# EPICS SNL sequencer program: dxp/branches/R3-0-branch/dxpApp/src/dxpMED.st
program dxpMED("P=13GE2:med:,DXP=dxp,MCA=mca,N_DETECTORS=16")

/*  This sequencer program works with dxp.db and dxpMED.db.
 *  It supports Copying PVs from the first DXP to all of the DXPs
 *  and multi-element MCA operations
 *
 *  Mark Rivers
 *  January 7, 2005
 *
 * This program must be compiled with the recursive option so that multiple copies
 * can run at once */
option +r;

/* Allow the program to start, even if not all assigned channels are connected.
 * This could be useful if dxpMED is running on a different ioc. */
option -c;

%%#include <stdlib.h>
%%#include <errlog.h>

#define MAX_DETECTORS 100
#define MAX_SCAS 16
/* MAX_ROIS must be defined as MAX_DETECTORS * MAX_SCAS.
   It can't be done in SNL because of syntax limitations. */
#define MAX_ROIS 1600

int i;
int j;
int k;
int chan;
int det;
int nDetectors;
int prevAcquiring;
int allDone;
char temp[100];

char *prefix;
char *dxp;
char *mca;

double  TriggerPeakingTime[MAX_DETECTORS];
assign  TriggerPeakingTime to {"","","","","","","","","","","","","","","","",
                       "","","","","","","","","","","","","","","",""};
int     CopyTriggerPeakingTime; assign CopyTriggerPeakingTime to "{P}CopyTriggerPeakingTime";
monitor CopyTriggerPeakingTime; evflag CopyTriggerPeakingTimeMon; sync CopyTriggerPeakingTime CopyTriggerPeakingTimeMon;

double  TriggerGapTime[MAX_DETECTORS];
assign  TriggerGapTime to {"","","","","","","","","","","","","","","","",
                        "","","","","","","","","","","","","","","",""};
int     CopyTriggerGapTime; assign CopyTriggerGapTime to "{P}CopyTriggerGapTime";
monitor CopyTriggerGapTime; evflag CopyTriggerGapTimeMon; sync CopyTriggerGapTime CopyTriggerGapTimeMon;

double  TriggerThreshold[MAX_DETECTORS];
assign  TriggerThreshold to {"","","","","","","","","","","","","","","","",
                      "","","","","","","","","","","","","","","",""};
int     CopyTriggerThreshold; assign CopyTriggerThreshold to "{P}CopyTriggerThreshold";
monitor CopyTriggerThreshold; evflag CopyTriggerThresholdMon; sync CopyTriggerThreshold CopyTriggerThresholdMon;

double  PeakingTime[MAX_DETECTORS];
assign  PeakingTime to {"","","","","","","","","","","","","","","","",
                  "","","","","","","","","","","","","","","",""};
int     CopyPeakingTime; assign CopyPeakingTime to "{P}CopyPeakingTime";
monitor CopyPeakingTime; evflag CopyPeakingTimeMon; sync CopyPeakingTime CopyPeakingTimeMon;

double  GapTime[MAX_DETECTORS];
assign  GapTime to {"","","","","","","","","","","","","","","","",
                   "","","","","","","","","","","","","","","",""};
int     CopyGapTime; assign CopyGapTime to "{P}CopyGapTime";
monitor CopyGapTime; evflag CopyGapTimeMon; sync CopyGapTime CopyGapTimeMon;

double  EnergyThreshold[MAX_DETECTORS];
assign  EnergyThreshold to {"","","","","","","","","","","","","","","","",
                      "","","","","","","","","","","","","","","",""};
int     CopyEnergyThreshold; assign CopyEnergyThreshold to "{P}CopyEnergyThreshold";
monitor CopyEnergyThreshold; evflag CopyEnergyThresholdMon; sync CopyEnergyThreshold CopyEnergyThresholdMon;

double  MaxWidth[MAX_DETECTORS];
assign  MaxWidth to {"","","","","","","","","","","","","","","","",
                      "","","","","","","","","","","","","","","",""};
int     CopyMaxWidth; assign CopyMaxWidth to "{P}CopyMaxWidth";
monitor CopyMaxWidth; evflag CopyMaxWidthMon; sync CopyMaxWidth CopyMaxWidthMon;

double  BaselineCutPercent[MAX_DETECTORS];
assign  BaselineCutPercent to {"","","","","","","","","","","","","","","","",
                         "","","","","","","","","","","","","","","",""};
int     CopyBaselineCutPercent; assign CopyBaselineCutPercent to "{P}CopyBaselineCutPercent";
monitor CopyBaselineCutPercent; evflag CopyBaselineCutPercentMon; sync CopyBaselineCutPercent CopyBaselineCutPercentMon;

double  BaselineCutEnable[MAX_DETECTORS];
assign  BaselineCutEnable to {"","","","","","","","","","","","","","","","",
                          "","","","","","","","","","","","","","","",""};
int     CopyBaselineCutEnable; assign CopyBaselineCutEnable to "{P}CopyBaselineCutEnable";
monitor CopyBaselineCutEnable; evflag CopyBaselineCutEnableMon; sync CopyBaselineCutEnable CopyBaselineCutEnableMon;

double  BaselineThreshold[MAX_DETECTORS];
assign  BaselineThreshold to {"","","","","","","","","","","","","","","","",
                        "","","","","","","","","","","","","","","",""};
int     CopyBaselineThreshold; assign CopyBaselineThreshold to "{P}CopyBaselineThreshold";
monitor CopyBaselineThreshold; evflag CopyBaselineThresholdMon; sync CopyBaselineThreshold CopyBaselineThresholdMon;

double  BaselineFilterLength[MAX_DETECTORS];
assign  BaselineFilterLength to {"","","","","","","","","","","","","","","","",
                     "","","","","","","","","","","","","","","",""};
int     CopyBaselineFilterLength; assign CopyBaselineFilterLength to "{P}CopyBaselineFilterLength";
monitor CopyBaselineFilterLength; evflag CopyBaselineFilterLengthMon; sync CopyBaselineFilterLength CopyBaselineFilterLengthMon;

double  PreampGain[MAX_DETECTORS];
assign  PreampGain to {"","","","","","","","","","","","","","","","",
                  "","","","","","","","","","","","","","","",""};
int     CopyPreampGain; assign CopyPreampGain to "{P}CopyPreampGain";
monitor CopyPreampGain; evflag CopyPreampGainMon; sync CopyPreampGain CopyPreampGainMon;

double  MaxEnergy[MAX_DETECTORS];
assign  MaxEnergy to {"","","","","","","","","","","","","","","","",
                 "","","","","","","","","","","","","","","",""};
int     CopyMaxEnergy; assign CopyMaxEnergy to "{P}CopyMaxEnergy";
monitor CopyMaxEnergy; evflag CopyMaxEnergyMon; sync CopyMaxEnergy CopyMaxEnergyMon;

double  ADCPercentRule[MAX_DETECTORS];
assign  ADCPercentRule to {"","","","","","","","","","","","","","","","",
                     "","","","","","","","","","","","","","","",""};
int     CopyADCPercentRule; assign CopyADCPercentRule to "{P}CopyADCPercentRule";
monitor CopyADCPercentRule; evflag CopyADCPercentRuleMon; sync CopyADCPercentRule CopyADCPercentRuleMon;

/*int     ReadDXP[MAX_DETECTORS];  */
/*assign  ReadDXP to {"","","","","","","","","","","","","","","","", */
/*                    "","","","","","","","","","","","","","","",""}; */
/*int     ReadDXPs; assign ReadDXPs to "{P}DoReadDXPs"; */
/*monitor ReadDXPs; evflag ReadDXPsMon; sync ReadDXPs ReadDXPsMon; */

int     ReadBaselineHistogram[MAX_DETECTORS];
assign  ReadBaselineHistogram to {"","","","","","","","","","","","","","","","",
                            "","","","","","","","","","","","","","","",""};
int     ReadBaselineHistograms; assign ReadBaselineHistograms to "{P}DoReadBaselineHistograms";
monitor ReadBaselineHistograms; evflag ReadBaselineHistogramsMon; sync ReadBaselineHistograms ReadBaselineHistogramsMon;

int     ReadTrace[MAX_DETECTORS];
assign  ReadTrace to {"","","","","","","","","","","","","","","","",
                         "","","","","","","","","","","","","","","",""};
int     ReadTraces; assign ReadTraces to "{P}DoReadTraces";
monitor ReadTraces; evflag ReadTracesMon; sync ReadTraces ReadTracesMon;

double  TraceTime[MAX_DETECTORS];
assign  TraceTime to {"","","","","","","","","","","","","","","","",
                         "","","","","","","","","","","","","","","",""};
double  TraceTimes; assign TraceTimes to "{P}TraceTimes";
monitor TraceTimes; evflag TraceTimesMon; sync TraceTimes TraceTimesMon;

int     TraceMode[MAX_DETECTORS];
assign  TraceMode to {"","","","","","","","","","","","","","","","",
                         "","","","","","","","","","","","","","","",""};
int     TraceModes; assign TraceModes to "{P}TraceModes";
monitor TraceModes; evflag TraceModesMon; sync TraceModes TraceModesMon;

int     ReadMCA[MAX_DETECTORS];
assign  ReadMCA to {"","","","","","","","","","","","","","","","",
                    "","","","","","","","","","","","","","","",""};
int     ReadMCAs; assign ReadMCAs to "{P}DoReadAll";
monitor ReadMCAs; evflag ReadMCAsMon; sync ReadMCAs ReadMCAsMon;
int     ReadMCAAll; assign ReadMCAAll to "";

int     statusMCA[MAX_DETECTORS];
assign  statusMCA to {"","","","","","","","","","","","","","","","",
                      "","","","","","","","","","","","","","","",""};
int     StatusMCAs; assign StatusMCAs to "{P}DoStatusAll";
monitor StatusMCAs; evflag StatusMCAsMon; sync StatusMCAs StatusMCAsMon;
int     statusMCAAll; assign statusMCAAll to "";

int     mcaAcquiring[MAX_DETECTORS];
assign  mcaAcquiring to {"","","","","","","","","","","","","","","","",
                         "","","","","","","","","","","","","","","",""};
monitor mcaAcquiring; evflag  mcaAcquiringMon; sync mcaAcquiring mcaAcquiringMon;
int     Acquiring; assign Acquiring to "";
monitor Acquiring; evflag AcquiringMon; sync Acquiring AcquiringMon;

double  mcaPresetReal[MAX_DETECTORS];
assign  mcaPresetReal to {"","","","","","","","","","","","","","","","",
                          "","","","","","","","","","","","","","","",""};
double  PresetReal; assign PresetReal to "{P}PresetReal";
monitor PresetReal; evflag PresetRealMon; sync PresetReal PresetRealMon;

double  mcaPresetLive[MAX_DETECTORS];
assign  mcaPresetLive to {"","","","","","","","","","","","","","","","",
                          "","","","","","","","","","","","","","","",""};
double  PresetLive; assign PresetLive to "{P}PresetLive";
monitor PresetLive; evflag PresetLiveMon; sync PresetLive PresetLiveMon;

double  mcaDeadTime[MAX_DETECTORS];
assign  mcaDeadTime to {"","","","","","","","","","","","","","","","",
                        "","","","","","","","","","","","","","","",""};
double  DeadTime; assign DeadTime to "{P}DeadTime";
evflag  DeadTimeMon; sync mcaDeadTime DeadTimeMon;

int     mcaROILow[MAX_ROIS];
assign  mcaROILow to {"","","","","","","","","","","","","","","","",
                      "","","","","","","","","","","","","","","","",
                      "","","","","","","","","","","","","","","","",
                      "","","","","","","","","","","","","","","","",
                      "","","","","","","","","","","","","","","","",
                      "","","","","","","","","","","","","","","","",
                      "","","","","","","","","","","","","","","","",
                      "","","","","","","","","","","","","","","","",
                      "","","","","","","","","","","","","","","","",
                      "","","","","","","","","","","","","","","","",
                      "","","","","","","","","","","","","","","","",
                      "","","","","","","","","","","","","","","","",
                      "","","","","","","","","","","","","","","","",
                      "","","","","","","","","","","","","","","","",
                      "","","","","","","","","","","","","","","","",
                      "","","","","","","","","","","","","","","","",
                      "","","","","","","","","","","","","","","","",
                      "","","","","","","","","","","","","","","","",
                      "","","","","","","","","","","","","","","","",
                      "","","","","","","","","","","","","","","","",
                      "","","","","","","","","","","","","","","","",
                      "","","","","","","","","","","","","","","","",
                      "","","","","","","","","","","","","","","","",
                      "","","","","","","","","","","","","","","","",
                      "","","","","","","","","","","","","","","","",
                      "","","","","","","","","","","","","","","","",
                      "","","","","","","","","","","","","","","","",
                      "","","","","","","","","","","","","","","","",
                      "","","","","","","","","","","","","","","","",
                      "","","","","","","","","","","","","","","","",
                      "","","","","","","","","","","","","","","","",
                      "","","","","","","","","","","","","","","",""};
monitor mcaROILow; evflag  mcaROILowMon; sync mcaROILow mcaROILowMon;

int    mcaROIHigh[MAX_ROIS];
assign mcaROIHigh to {"","","","","","","","","","","","","","","","",
                      "","","","","","","","","","","","","","","","",
                      "","","","","","","","","","","","","","","","",
                      "","","","","","","","","","","","","","","","",
                      "","","","","","","","","","","","","","","","",
                      "","","","","","","","","","","","","","","","",
                      "","","","","","","","","","","","","","","","",
                      "","","","","","","","","","","","","","","","",
                      "","","","","","","","","","","","","","","","",
                      "","","","","","","","","","","","","","","","",
                      "","","","","","","","","","","","","","","","",
                      "","","","","","","","","","","","","","","","",
                      "","","","","","","","","","","","","","","","",
                      "","","","","","","","","","","","","","","","",
                      "","","","","","","","","","","","","","","","",
                      "","","","","","","","","","","","","","","","",
                      "","","","","","","","","","","","","","","","",
                      "","","","","","","","","","","","","","","","",
                      "","","","","","","","","","","","","","","","",
                      "","","","","","","","","","","","","","","","",
                      "","","","","","","","","","","","","","","","",
                      "","","","","","","","","","","","","","","","",
                      "","","","","","","","","","","","","","","","",
                      "","","","","","","","","","","","","","","","",
                      "","","","","","","","","","","","","","","","",
                      "","","","","","","","","","","","","","","","",
                      "","","","","","","","","","","","","","","","",
                      "","","","","","","","","","","","","","","","",
                      "","","","","","","","","","","","","","","","",
                      "","","","","","","","","","","","","","","","",
                      "","","","","","","","","","","","","","","","",
                      "","","","","","","","","","","","","","","",""};
monitor mcaROIHigh; evflag  mcaROIHighMon; sync mcaROIHigh mcaROIHighMon;

int     dxpSCALow[MAX_ROIS];
assign  dxpSCALow to {"","","","","","","","","","","","","","","","",
                      "","","","","","","","","","","","","","","","",
                      "","","","","","","","","","","","","","","","",
                      "","","","","","","","","","","","","","","","",
                      "","","","","","","","","","","","","","","","",
                      "","","","","","","","","","","","","","","","",
                      "","","","","","","","","","","","","","","","",
                      "","","","","","","","","","","","","","","","",
                      "","","","","","","","","","","","","","","","",
                      "","","","","","","","","","","","","","","","",
                      "","","","","","","","","","","","","","","","",
                      "","","","","","","","","","","","","","","","",
                      "","","","","","","","","","","","","","","","",
                      "","","","","","","","","","","","","","","","",
                      "","","","","","","","","","","","","","","","",
                      "","","","","","","","","","","","","","","","",
                      "","","","","","","","","","","","","","","","",
                      "","","","","","","","","","","","","","","","",
                      "","","","","","","","","","","","","","","","",
                      "","","","","","","","","","","","","","","","",
                      "","","","","","","","","","","","","","","","",
                      "","","","","","","","","","","","","","","","",
                      "","","","","","","","","","","","","","","","",
                      "","","","","","","","","","","","","","","","",
                      "","","","","","","","","","","","","","","","",
                      "","","","","","","","","","","","","","","","",
                      "","","","","","","","","","","","","","","","",
                      "","","","","","","","","","","","","","","","",
                      "","","","","","","","","","","","","","","","",
                      "","","","","","","","","","","","","","","","",
                      "","","","","","","","","","","","","","","","",
                      "","","","","","","","","","","","","","","",""};

int    dxpSCAHigh[MAX_ROIS];
assign dxpSCAHigh to {"","","","","","","","","","","","","","","","",
                      "","","","","","","","","","","","","","","","",
                      "","","","","","","","","","","","","","","","",
                      "","","","","","","","","","","","","","","","",
                      "","","","","","","","","","","","","","","","",
                      "","","","","","","","","","","","","","","","",
                      "","","","","","","","","","","","","","","","",
                      "","","","","","","","","","","","","","","","",
                      "","","","","","","","","","","","","","","","",
                      "","","","","","","","","","","","","","","","",
                      "","","","","","","","","","","","","","","","",
                      "","","","","","","","","","","","","","","","",
                      "","","","","","","","","","","","","","","","",
                      "","","","","","","","","","","","","","","","",
                      "","","","","","","","","","","","","","","","",
                      "","","","","","","","","","","","","","","","",
                      "","","","","","","","","","","","","","","","",
                      "","","","","","","","","","","","","","","","",
                      "","","","","","","","","","","","","","","","",
                      "","","","","","","","","","","","","","","","",
                      "","","","","","","","","","","","","","","","",
                      "","","","","","","","","","","","","","","","",
                      "","","","","","","","","","","","","","","","",
                      "","","","","","","","","","","","","","","","",
                      "","","","","","","","","","","","","","","","",
                      "","","","","","","","","","","","","","","","",
                      "","","","","","","","","","","","","","","","",
                      "","","","","","","","","","","","","","","","",
                      "","","","","","","","","","","","","","","","",
                      "","","","","","","","","","","","","","","","",
                      "","","","","","","","","","","","","","","","",
                      "","","","","","","","","","","","","","","",""};

int AcquireBusy; assign AcquireBusy to "{P}AcquireBusy";

ss dxp_control {
    state init {
        when() {
            /* We set the following event flags to force these modes and
               labels to be set correctly initially */
            prefix = macValueGet("P");
            dxp = macValueGet("DXP");
            mca = macValueGet("MCA");
            nDetectors = atoi(macValueGet("N_DETECTORS"));
            if ((nDetectors <= 0) || (nDetectors > MAX_DETECTORS)) {
              printf ("N_DETECTORS is illegal.\n");
              nDetectors = 0;
            }
            if (MAX_ROIS != (MAX_DETECTORS * MAX_SCAS)) {
              printf ("N_DETECTORS, MAX_SCAS and MAX_ROIS are inconsistent.\n");
              nDetectors = 0;
            }
            for (i=0; i<nDetectors; i++) {
               det = i+1;
               sprintf(temp, "%s%s%d:TriggerPeakingTime", prefix, dxp, det);
               pvAssign(TriggerPeakingTime[i], temp);
               sprintf(temp, "%s%s%d:TriggerGapTime", prefix, dxp, det);
               pvAssign(TriggerGapTime[i], temp);
               sprintf(temp, "%s%s%d:TriggerThreshold", prefix, dxp, det);
               pvAssign(TriggerThreshold[i], temp);
               sprintf(temp, "%s%s%d:PeakingTime", prefix, dxp, det);
               pvAssign(PeakingTime[i], temp);
               sprintf(temp, "%s%s%d:GapTime", prefix, dxp, det);
               pvAssign(GapTime[i], temp);
               sprintf(temp, "%s%s%d:EnergyThreshold", prefix, dxp, det);
               pvAssign(EnergyThreshold[i], temp);
               sprintf(temp, "%s%s%d:MaxWidth", prefix, dxp, det);
               pvAssign(MaxWidth[i], temp);
               sprintf(temp, "%s%s%d:BaselineCutPercent", prefix, dxp, det);
               pvAssign(BaselineCutPercent[i], temp);
               sprintf(temp, "%s%s%d:BaselineCutEnable", prefix, dxp, det);
               pvAssign(BaselineCutEnable[i], temp);
               sprintf(temp, "%s%s%d:BaselineThreshold", prefix, dxp, det);
               pvAssign(BaselineThreshold[i], temp);
               sprintf(temp, "%s%s%d:BaselineFilterLength", prefix, dxp, det);
               pvAssign(BaselineFilterLength[i], temp);
               sprintf(temp, "%s%s%d:PreampGain", prefix, dxp, det);
               pvAssign(PreampGain[i], temp);
               sprintf(temp, "%s%s%d:MaxEnergy", prefix, dxp, det);
               pvAssign(MaxEnergy[i], temp);
               sprintf(temp, "%s%s%d:ADCPercentRule", prefix, dxp, det);
               pvAssign(ADCPercentRule[i], temp);
/*               sprintf(temp, "%s%s%d:ReadParams.PROC", prefix, dxp, det); */
/*               pvAssign(ReadDXP[i], temp); */
               sprintf(temp, "%s%s%d:BaselineHistogram.PROC", prefix, dxp, det);
               pvAssign(ReadBaselineHistogram[i], temp);
               sprintf(temp, "%s%s%d:TraceData.PROC", prefix, dxp, det);
               pvAssign(ReadTrace[i], temp);
               sprintf(temp, "%s%s%d:TraceTime", prefix, dxp, det);
               pvAssign(TraceTime[i], temp);
               sprintf(temp, "%s%s%d:TraceMode", prefix, dxp, det);
               pvAssign(TraceMode[i], temp);
               sprintf(temp, "%s%s%d.READ", prefix, mca, det);
               pvAssign(ReadMCA[i], temp);
               sprintf(temp, "%s%s%d.PROC", prefix, mca, det);
               pvAssign(statusMCA[i], temp);
               sprintf(temp, "%s%s%d.ACQG", prefix, mca, det);
               pvAssign(mcaAcquiring[i], temp);
               sprintf(temp, "%s%s%d.PRTM", prefix, mca, det);
               pvAssign(mcaPresetReal[i], temp);
               sprintf(temp, "%s%s%d.PLTM", prefix, mca, det);
               pvAssign(mcaPresetLive[i], temp);
               sprintf(temp, "%s%s%d.IDTIM", prefix, mca, det);
               pvAssign(mcaDeadTime[i], temp);
               pvMonitor(mcaDeadTime[i]);
/*
               for (j=0; j<MAX_SCAS; j++) {
                   k = i*MAX_SCAS + j;
                   sprintf(temp, "%s%s%d.R%iLO", prefix, mca, det, j);
                   pvAssign(mcaROILow[k], temp);
                   pvMonitor(mcaROILow[k]);
                   sprintf(temp, "%s%s%d.R%iHI", prefix, mca, det, j);
                   pvAssign(mcaROIHigh[k], temp);
                   pvMonitor(mcaROIHigh[k]);
                   sprintf(temp, "%s%s%d.SCA%i_LO", prefix, dxp, det, j);
                   pvAssign(dxpSCALow[k], temp);
                   sprintf(temp, "%s%s%d.SCA%i_HI", prefix, dxp, det, j);
                   pvAssign(dxpSCAHigh[k], temp);
               }
*/
           }
           sprintf(temp, "%s%sAll.PROC", prefix, mca);
           pvAssign(statusMCAAll, temp);
           sprintf(temp, "%s%sAll.READ", prefix, mca);
           pvAssign(ReadMCAAll, temp);
           sprintf(temp, "%s%sAll.ACQG", prefix, mca);
           pvAssign(Acquiring, temp);
           prevAcquiring = Acquiring;
        } state waitConnected
    }
    state waitConnected {

        when (nDetectors <= 0) {
          printf (">>>>>>>>>>>>>> dxpMED is dead. <<<<<<<<<<<<<<\n");
        } state dead

        when (pvAssignCount () == pvConnectCount ()) {
          printf ("dxpMED: All channels connected.\n");
        } state monitor_changes

    }
    state dead {
      when (delay (3600.0)) {
      } state dead
    }

    state monitor_changes {

        when (pvAssignCount () != pvConnectCount ()) {
          printf ("dxpMED: Not all channels connected.\n");
        } state waitConnected

        when(efTestAndClear(CopyTriggerPeakingTimeMon) && (CopyTriggerPeakingTime == 1)) {
            pvGet(TriggerPeakingTime[0]);
            for (i=0; i<nDetectors; i++) {
                TriggerPeakingTime[i] = TriggerPeakingTime[0];
                pvPut(TriggerPeakingTime[i]);
            }
            CopyTriggerPeakingTime = 0;
            pvPut(CopyTriggerPeakingTime);
        } state monitor_changes

        when(efTestAndClear(CopyTriggerGapTimeMon) && (CopyTriggerGapTime == 1)) {
            pvGet(TriggerGapTime[0]);
            for (i=0; i<nDetectors; i++) {
                TriggerGapTime[i] = TriggerGapTime[0];
                pvPut(TriggerGapTime[i]);
            }
            CopyTriggerGapTime = 0;
            pvPut(CopyTriggerGapTime);
        } state monitor_changes

        when(efTestAndClear(CopyTriggerThresholdMon) && (CopyTriggerThreshold == 1)) {
            pvGet(TriggerThreshold[0]);
            for (i=0; i<nDetectors; i++) {
                TriggerThreshold[i] = TriggerThreshold[0];
                pvPut(TriggerThreshold[i]);
            }
            CopyTriggerThreshold = 0;
            pvPut(CopyTriggerThreshold);
        } state monitor_changes

        when(efTestAndClear(CopyPeakingTimeMon) && (CopyPeakingTime == 1)) {
            pvGet(PeakingTime[0]);
            for (i=0; i<nDetectors; i++) {
                PeakingTime[i] = PeakingTime[0];
                pvPut(PeakingTime[i]);
            }
            CopyPeakingTime = 0;
            pvPut(CopyPeakingTime);
        } state monitor_changes

        when(efTestAndClear(CopyGapTimeMon) && (CopyGapTime == 1)) {
            pvGet(GapTime[0]);
            for (i=0; i<nDetectors; i++) {
                GapTime[i] = GapTime[0];
                pvPut(GapTime[i]);
            }
            CopyGapTime = 0;
            pvPut(CopyGapTime);
        } state monitor_changes

        when(efTestAndClear(CopyEnergyThresholdMon) && (CopyEnergyThreshold == 1)) {
            pvGet(EnergyThreshold[0]);
            for (i=0; i<nDetectors; i++) {
                EnergyThreshold[i] = EnergyThreshold[0];
                pvPut(EnergyThreshold[i]);
            }
            CopyEnergyThreshold = 0;
            pvPut(CopyEnergyThreshold);
        } state monitor_changes

        when(efTestAndClear(CopyMaxWidthMon) && (CopyMaxWidth == 1)) {
            pvGet(MaxWidth[0]);
            for (i=0; i<nDetectors; i++) {
                MaxWidth[i] = MaxWidth[0];
                pvPut(MaxWidth[i]);
            }
            CopyMaxWidth = 0;
            pvPut(CopyMaxWidth);
        } state monitor_changes

        when(efTestAndClear(CopyBaselineCutPercentMon) && (CopyBaselineCutPercent == 1)) {
            pvGet(BaselineCutPercent[0]);
            for (i=0; i<nDetectors; i++) {
                BaselineCutPercent[i] = BaselineCutPercent[0];
                pvPut(BaselineCutPercent[i]);
            }
            CopyBaselineCutPercent = 0;
            pvPut(CopyBaselineCutPercent);
        } state monitor_changes

        when(efTestAndClear(CopyBaselineCutEnableMon) && (CopyBaselineCutEnable == 1)) {
            pvGet(BaselineCutEnable[0]);
            for (i=0; i<nDetectors; i++) {
                BaselineCutEnable[i] = BaselineCutEnable[0];
                pvPut(BaselineCutEnable[i]);
            }
            CopyBaselineCutEnable = 0;
            pvPut(CopyBaselineCutEnable);
        } state monitor_changes

        when(efTestAndClear(CopyBaselineThresholdMon) && (CopyBaselineThreshold == 1)) {
            pvGet(BaselineThreshold[0]);
            for (i=0; i<nDetectors; i++) {
                BaselineThreshold[i] = BaselineThreshold[0];
                pvPut(BaselineThreshold[i]);
            }
            CopyBaselineThreshold = 0;
            pvPut(CopyBaselineThreshold);
        } state monitor_changes

        when(efTestAndClear(CopyBaselineFilterLengthMon) && (CopyBaselineFilterLength == 1)) {
            pvGet(BaselineFilterLength[0]);
            for (i=0; i<nDetectors; i++) {
                BaselineFilterLength[i] = BaselineFilterLength[0];
                pvPut(BaselineFilterLength[i]);
            }
            CopyBaselineFilterLength = 0;
            pvPut(CopyBaselineFilterLength);
        } state monitor_changes

        when(efTestAndClear(CopyPreampGainMon) && (CopyPreampGain == 1)) {
            pvGet(PreampGain[0]);
            for (i=0; i<nDetectors; i++) {
                PreampGain[i] = PreampGain[0];
                pvPut(PreampGain[i]);
            }
            CopyPreampGain = 0;
            pvPut(CopyPreampGain);
        } state monitor_changes

        when(efTestAndClear(CopyMaxEnergyMon) && (CopyMaxEnergy == 1)) {
            pvGet(MaxEnergy[0]);
            for (i=0; i<nDetectors; i++) {
                MaxEnergy[i] = MaxEnergy[0];
                pvPut(MaxEnergy[i]);
            }
            CopyMaxEnergy = 0;
            pvPut(CopyMaxEnergy);
        } state monitor_changes

        when(efTestAndClear(CopyADCPercentRuleMon) && (CopyADCPercentRule == 1)) {
            pvGet(ADCPercentRule[0]);
            for (i=0; i<nDetectors; i++) {
                ADCPercentRule[i] = ADCPercentRule[0];
                pvPut(ADCPercentRule[i]);
            }
            CopyADCPercentRule = 0;
            pvPut(CopyADCPercentRule);
        } state monitor_changes

/*        when(efTestAndClear(ReadDXPsMon) && (ReadDXPs == 1)) {
            for (i=0; i<nDetectors; i++) {
                ReadDXP[i] = 1;
                pvPut(ReadDXP[i]);
            }
            ReadDXPs = 0;
            pvPut(ReadDXPs);
        } state monitor_changes  */

        when(efTestAndClear(ReadBaselineHistogramsMon) && (ReadBaselineHistograms == 1)) {
            for (i=0; i<nDetectors; i++) {
                ReadBaselineHistogram[i] = 1;
                pvPut(ReadBaselineHistogram[i]);
            }
            ReadBaselineHistograms = 0;
            pvPut(ReadBaselineHistograms);
        } state monitor_changes

        when(efTestAndClear(ReadTracesMon) && (ReadTraces == 1)) {
            for (i=0; i<nDetectors; i++) {
                ReadTrace[i] = 1;
                pvPut(ReadTrace[i]);
            }
            ReadTraces = 0;
            pvPut(ReadTraces);
        } state monitor_changes

        when(efTestAndClear(TraceTimesMon)) {
            for (i=0; i<nDetectors; i++) {
                TraceTime[i] = TraceTimes;
                pvPut(TraceTime[i]);
            }
        } state monitor_changes

        when(efTestAndClear(TraceModesMon)) {
            for (i=0; i<nDetectors; i++) {
                TraceMode[i] = TraceModes;
                pvPut(TraceMode[i]);
            }
        } state monitor_changes

        when(efTestAndClear(ReadMCAsMon) && (ReadMCAs == 1)) {
            /* printf("dxpMED: Read MCAs\n"); */
            for (i=0; i<nDetectors; i++) {
                ReadMCA[i] = 1;
                pvPut(ReadMCA[i]);
            }
            ReadMCAAll = 1;
            pvPut(ReadMCAAll);
            ReadMCAs = 0;
            pvPut(ReadMCAs);
        } state monitor_changes

        when(efTestAndClear(StatusMCAsMon) && (StatusMCAs == 1)) {
            /* printf("dxpMED: Read MCA status\n"); */
            for (i=0; i<nDetectors; i++) {
                statusMCA[i] = 1;
                pvPut(statusMCA[i]);
            }
            statusMCAAll = 1;
            pvPut(statusMCAAll);
            StatusMCAs = 0;
            pvPut(StatusMCAs);
        } state monitor_changes

        when(efTestAndClear(AcquiringMon)) {
            /* printf("dxpMED: Acquiring=%d, prevAcquiring=%d\n", Acquiring, prevAcquiring); */
            /* On the transition from Acquiring=1 to 0 clear the AcquireBusy record */
            if ((Acquiring == 0) && (prevAcquiring == 1)) {
               AcquireBusy = 0;
               pvPut(AcquireBusy);
            }
            prevAcquiring = Acquiring;
        } state monitor_changes

        when(efTestAndClear(mcaAcquiringMon)) {
            /* Transition on one or more mcaAcquiring status, wait 10msec for mcaAll to also change */
            allDone = 1;
            for (i=0; i<nDetectors; i++) {
                if (mcaAcquiring[i]) allDone = 0;
            }
            /* If all individual MCAs are done, but mcaAll is not done, then force Read on mcaAll */
            if (allDone && Acquiring) {
               ReadMCAAll = 1;
               pvPut(ReadMCAAll);
            }
        } state monitor_changes

        when(efTestAndClear(PresetRealMon)) {
            for (i=0; i<nDetectors; i++) {
                mcaPresetReal[i] = PresetReal;
                pvPut(mcaPresetReal[i]);
            }
        } state monitor_changes

        when(efTestAndClear(PresetLiveMon)) {
            for (i=0; i<nDetectors; i++) {
                mcaPresetLive[i] = PresetLive;
                pvPut(mcaPresetLive[i]);
            }
        } state monitor_changes

        when(efTestAndClear(DeadTimeMon)) {
            DeadTime = 0.;
            for (i=0; i<nDetectors; i++) {
                if (mcaDeadTime[i] > DeadTime) DeadTime = mcaDeadTime[i];
            }
            pvPut(DeadTime);
        } state monitor_changes

        /* Copy ROIs to SCAs */
 /*
        when(efTestAndClear(mcaROILowMon) || efTestAndClear(mcaROIHighMon)) {
            for (i=0; i<nDetectors; i++) {
                for (j=0; j<MAX_SCAS; j++) {
                    k = i*MAX_SCAS + j;
                    chan = mcaROILow[k];
                    if (chan < 0) chan = 0;
                    dxpSCALow[k] = chan;
                    pvPut(dxpSCALow[k]);
                    chan = mcaROIHigh[k];
                    if (chan < 0) chan = 0;
                    dxpSCAHigh[k] = chan;
                    pvPut(dxpSCAHigh[k]);
                }
            }
        } state monitor_changes
*/

   }
}
